# B&R Automation Studio project automationLearning
Automation Studio 4.9

## Configuration MirUnitTest

CPU X20CP0484, AutomationRuntime 6.0.2, Build 11.3.0, Vc 6.0.0

### Hardware
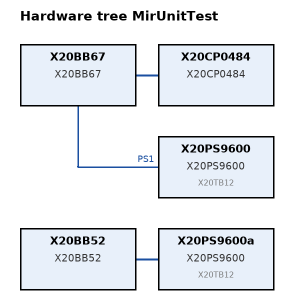
```
X20BB52 : X20BB52 v1.2.0.0
X20BB67 : X20BB67 v1.3.0.0
X20CP0484 : X20CP0484 v1.8.1.0  [SL -> X20BB67.SL1]
  TimerDeviceType = SWIOTIMER
  Cyclic1Duration = 10000
  Cyclic1Tolerance = 10000
  Cyclic2Duration = 20000
  Cyclic2Tolerance = 20000
  Cyclic3Duration = 50000
  Cyclic3Tolerance = 50000
  Cyclic4Duration = 100000
  Cyclic4Tolerance = 100000
  Cyclic5Duration = 200000
  Cyclic5Tolerance = 200000
  Cyclic6Duration = 500000
  Cyclic6Tolerance = 500000
  Cyclic7Duration = 1000000
  Cyclic7Tolerance = 1000000
  Cyclic8Duration = 10000
  Cyclic8Tolerance = 30000000
  FileDevice1
  FileDeviceName1 = USER
  FileDevicePath1 = USER_PATH
X20PS9600 : X20PS9600 v1.6.2.0  [PS -> X20BB67.PS1; SS1 -> X20TB12.SS]
X20PS9600a : X20PS9600 v1.6.2.0  [PS -> X20BB52.PS1; SS1 -> X20TB12a.SS]
X20TB12 : X20TB12 v1.0.0.0
X20TB12a : X20TB12 v1.0.0.0
```

## Configuration Mir_config1

CPU X20CP0484-1, AutomationRuntime 6.0.2, Build 11.3.0, Vc 6.0.0

### Task classes (Cpu.sw)
```
Cyclic#4 (cycle 100000 us, tolerance 100000 us):
  MirValveEx <- MirValveExample.prg
  HMI <- HMI.prg
  MirValveE1 <- MirValveExampleST.prg
Libraries: Valve
```

### Hardware
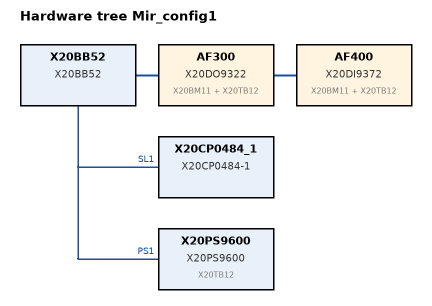
```
AF300 : X20DO9322 v1.6.2.0  [SS1 -> X20TB12a.SS; SL -> X20BM11.SL1]
AF400 : X20DI9372 v1.6.1.0  [SS1 -> X20TB12b.SS; SL -> X20BM11a.SL1]
X20BB52 : X20BB52 v1.2.0.0
  Connector IF6:
    CycleTime = 2000
X20BM11 : X20BM11 v1.1.0.0  [X2X1 -> X20BB52.IF6]
X20BM11a : X20BM11 v1.1.0.0  [X2X1 -> X20BM11.X2X2]
X20CP0484_1 : X20CP0484-1 v1.8.1.0  [SL -> X20BB52.SL1]
  Connector IF2:
    ActivateDevice = 1
  ConfigurationID = Mir_Mir_config1
  Simulation = 1
  TimerDeviceType = SWIOTIMER
  Cyclic1Duration = 10000
  Cyclic1Tolerance = 10000
  Cyclic2Duration = 20000
  Cyclic2Tolerance = 20000
  Cyclic3Duration = 50000
  Cyclic3Tolerance = 50000
  Cyclic4Duration = 100000
  Cyclic4Tolerance = 100000
  Cyclic5Duration = 200000
  Cyclic5Tolerance = 200000
  Cyclic6Duration = 500000
  Cyclic6Tolerance = 500000
  Cyclic7Duration = 1000000
  Cyclic7Tolerance = 1000000
  Cyclic8Duration = 10000
  Cyclic8Tolerance = 30000000
  FileDevice1
  FileDeviceName1 = USER
  FileDevicePath1 = USER_PATH
X20PS9600 : X20PS9600 v1.6.2.0  [PS -> X20BB52.PS1; SS1 -> X20TB12.SS]
X20TB12 : X20TB12 v1.0.0.0
X20TB12a : X20TB12 v1.0.0.0
X20TB12b : X20TB12 v1.0.0.0
```

### IoMap.iom - X20CP0484_1/IoMap.iom
```iecst
VAR_CONFIG
	::gValves.HV_1.cmd_out AT %QX."AF300".DigitalOutput01;
END_VAR
```

## Logical view

Binary libraries used (declarations not repeated): operator, runtime, AsIecCon, astime

### Package Logical/Libraries - Global libraries

### Library Logical/Libraries/MirLib (IEC)

#### Valve_on_off.fbd
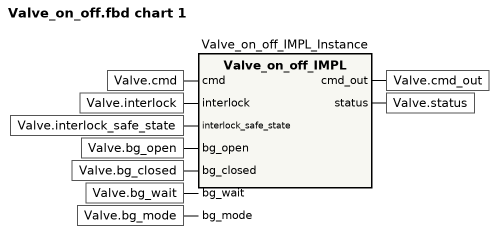
Diagram, in the editor's own instruction-list form stored in the file:
```il
FUNCTION_BLOCK Valve_on_off

{NetworkNumber := 1}
LD Valve.cmd
ST Valve_on_off_IMPL_Instance.cmd
LD Valve.interlock
ST Valve_on_off_IMPL_Instance.interlock
LD Valve.interlock_safe_state
ST Valve_on_off_IMPL_Instance.interlock_safe_state
LD Valve.bg_open
ST Valve_on_off_IMPL_Instance.bg_open
LD Valve.bg_closed
ST Valve_on_off_IMPL_Instance.bg_closed
LD Valve.bg_wait
ST Valve_on_off_IMPL_Instance.bg_wait
LD Valve.bg_mode
ST Valve_on_off_IMPL_Instance.bg_mode
CAL Valve_on_off_IMPL_Instance
LD Valve_on_off_IMPL_Instance.cmd_out
ST Valve.cmd_out
LD Valve_on_off_IMPL_Instance.status
ST Valve.status

END_FUNCTION_BLOCK
```

#### Types.typ - Exported data types
```iecst
TYPE
	bg_expected_enum :
		(
		BG_EXPECTED_OPEN := 0,
		BG_EXPECTED_CLOSED := 1
		);
	limit_switch_mode_enum :
		(
		BG_NONE := 0,
		BG_BOTH := 1,
		BG_OPEN := 2,
		BG_CLOSED := 3
		);
	valve_error_enum :
		(
		NONE := 0,
		TIMEOUT_OPENING := 1,
		TIMEOUT_CLOSING := 2,
		UNEXPECTED_CLOSED := 3,
		UNEXPECTED_OPEN := 4,
		BOTH_FEEDBACK := 5,
		NO_FEEDBACK := 6
		);
	valve_position_enum :
		(
		UNKNOWN := 0,
		CLOSED := 1,
		OPEN := 2,
		INTERMEDIATE := 3
		);
	valve_state_enum :
		(
		OK := 0,
		INTERLOCKED := 1,
		SUPERVISING := 2,
		ERROR := 3
		);
	valve_status_typ : 	STRUCT
		position : valve_position_enum;
		error : valve_error_enum;
		state : valve_state_enum;
	END_STRUCT;
	valve_typ : 	STRUCT
		cmd : BOOL;
		cmd_out : BOOL;
		interlock_safe_state : BOOL;
		status : valve_status_typ;
		interlock : BOOL;
		bg_closed : BOOL;
		bg_open : BOOL;
		bg_wait : TIME;
		bg_mode : limit_switch_mode_enum;
	END_STRUCT;
END_TYPE
```

#### MirLib.fun - Exported functions and function blocks
```iecst
{REDUND_ERROR} FUNCTION_BLOCK Valve_on_off_IMPL (*TODO: Add your comment here*) (*$GROUP=Miro,$CAT=User,$GROUPICON=User.png,$CATICON=User.png*)
	VAR_INPUT
		cmd : {REDUND_UNREPLICABLE} BOOL;
	END_VAR
	VAR_OUTPUT
		cmd_out : BOOL;
	END_VAR
	VAR
		cmd_rising_edge : BOOL;
		cmd_falling_edge : BOOL;
		cmd_changed : BOOL;
		cmd_previous : BOOL;
	END_VAR
	VAR_INPUT
		interlock : BOOL;
		interlock_safe_state : BOOL;
	END_VAR
	VAR
		supervision_active : BOOL;
	END_VAR
	VAR_OUTPUT
		status : valve_status_typ;
	END_VAR
	VAR_INPUT
		bg_open : BOOL; (*Limnit switch for open position*)
		bg_closed : BOOL; (*Limit switch for closed position*)
		bg_wait : TIME;
		bg_mode : limit_switch_mode_enum; (*Limit switch mode*)
	END_VAR
	VAR
		bg_expected_state : bg_expected_enum;
		bg_error : BOOL;
		ElapsedTimer : MirElapsedTimer;
	END_VAR
END_FUNCTION_BLOCK

{REDUND_ERROR} FUNCTION_BLOCK Valve_on_off (*TODO: Add your comment here*) (*$GROUP=User,$CAT=User,$GROUPICON=User.png,$CATICON=User.png*)
	VAR_IN_OUT
		Valve : valve_typ;
	END_VAR
	VAR
		Valve_on_off_IMPL_Instance : Valve_on_off_IMPL;
	END_VAR
END_FUNCTION_BLOCK

{REDUND_ERROR} FUNCTION_BLOCK MirElapsedTimer (*TODO: Add your comment here*) (*$GROUP=User,$CAT=User,$GROUPICON=User.png,$CATICON=User.png*)
	VAR_INPUT
		Enable : {REDUND_UNREPLICABLE} BOOL;
		Delay : TIME;
	END_VAR
	VAR_OUTPUT
		Elapsed : TIME;
		Out : BOOL;
	END_VAR
	VAR
		last_cycle_time : TIME;
		delta_time : TIME;
		cur_time : TIME;
		timer_initialized : BOOL;
	END_VAR
END_FUNCTION_BLOCK
```

#### Valve_on_off_IMPL.st
```iecst
FUNCTION_BLOCK Valve_on_off_IMPL
	ElapsedTimer();
	// RISIGN EDGE OR FALLINH CHECK
	IF cmd = TRUE AND cmd_previous = FALSE THEN
		cmd_rising_edge := TRUE;
		ElapsedTimer.Enable := FALSE;
		bg_error := FALSE;
	ELSE
		cmd_rising_edge := FALSE;
	END_IF;

	IF cmd = FALSE AND cmd_previous = TRUE THEN
		cmd_falling_edge := TRUE;
		ElapsedTimer.Enable := FALSE;
		bg_error := FALSE;
	ELSE
		cmd_falling_edge := FALSE;
	END_IF;

	IF interlock = FALSE THEN ACT_UpdateCmdOut;
	ELSE
		cmd_out := interlock_safe_state;
	END_IF;

	// Handle rising edge
	IF cmd_rising_edge THEN
		CASE bg_mode OF
			BG_NONE:
				// No supervision needed

			BG_BOTH, BG_OPEN:
				ElapsedTimer.Delay := bg_wait;
				ElapsedTimer.Enable := TRUE;
				supervision_active := TRUE;
				bg_expected_state := BG_EXPECTED_OPEN; // Expecting valve to open

			BG_CLOSED:
			// No supervision needed
		END_CASE;
	END_IF;

	// Handle falling edge
	IF cmd_falling_edge THEN
		CASE bg_mode OF
			BG_NONE:
				// No supervision needed
			BG_BOTH, BG_CLOSED:
				ElapsedTimer.Delay := bg_wait;
				ElapsedTimer.Enable := TRUE;
				supervision_active := TRUE;
				bg_expected_state := BG_EXPECTED_CLOSED;

			BG_OPEN:
			// No supervision needed
		END_CASE;
	END_IF;

	// Supervision logic
	IF supervision_active THEN
		CASE bg_mode OF
			BG_BOTH:
				IF (bg_expected_state = BG_EXPECTED_OPEN AND bg_open AND NOT bg_closed) OR
					(bg_expected_state = BG_EXPECTED_CLOSED AND bg_closed AND NOT bg_open) THEN
					supervision_active := FALSE;
					ElapsedTimer.Enable := FALSE;
					bg_error := FALSE;
				END_IF;

			BG_OPEN:
				IF bg_expected_state = BG_EXPECTED_OPEN AND bg_open THEN
					supervision_active := FALSE;
					ElapsedTimer.Enable := FALSE;
					bg_error := FALSE;
				END_IF;

			BG_CLOSED:
				IF bg_expected_state = BG_EXPECTED_CLOSED AND bg_closed THEN
					supervision_active := FALSE;
					ElapsedTimer.Enable := FALSE;
					bg_error := FALSE;
				END_IF;
		END_CASE;

		IF ElapsedTimer.Out THEN
			bg_error := TRUE;
			supervision_active := FALSE;
			ElapsedTimer.Enable := FALSE;
		END_IF;
	END_IF;

	// Continuous monitoring after successful supervision
	IF NOT supervision_active AND NOT bg_error THEN
		CASE bg_mode OF
			BG_BOTH:
				IF cmd_out AND (NOT bg_open OR bg_closed) THEN
					bg_error := TRUE;
				ELSIF NOT cmd_out AND (bg_open OR NOT bg_closed) THEN
					bg_error := TRUE;
				END_IF;
			BG_OPEN:
				IF cmd_out AND NOT bg_open THEN
					bg_error := TRUE;
				END_IF;
			BG_CLOSED:
				IF NOT cmd_out AND NOT bg_closed THEN
					bg_error := TRUE;
				END_IF;
		END_CASE;
	END_IF;
	ACT_UpdateValveStatus;
	cmd_previous := cmd;
END_FUNCTION_BLOCK
```

#### ACT_UpdateCmdOut.st
```iecst
ACTION ACT_UpdateCmdOut:
	IF cmd = TRUE THEN
		cmd_out := TRUE;
	ELSE
		cmd_out := FALSE;
	END_IF;

END_ACTION
```

#### MirElapsedTimer.st
```iecst
(* TODO: Add your comment here *)
FUNCTION_BLOCK MirElapsedTimer
	IF Enable THEN
		IF NOT timer_initialized THEN
			last_cycle_time := clock_ms();
			Elapsed := T#0ms;
			timer_initialized := TRUE;
		ELSE
			cur_time := clock_ms();
			delta_time := cur_time - last_cycle_time;
			last_cycle_time := cur_time;
			Elapsed := Elapsed + delta_time;
		END_IF;
		IF Elapsed >= Delay THEN
			Out := TRUE;
		END_IF;
	ELSE
		Out := FALSE;
		Elapsed := T#0ms;
		timer_initialized := FALSE;
	END_IF;
END_FUNCTION_BLOCK
```

#### ACT_UpdateValveStatus.st
```iecst
ACTION ACT_UpdateValveStatus:

	CASE bg_mode OF
		BG_BOTH:
			IF bg_open AND NOT bg_closed THEN
				status.position := OPEN;
			ELSIF NOT bg_open AND bg_closed THEN
				status.position := CLOSED;
			ELSIF bg_open AND bg_closed THEN
				status.position := INTERMEDIATE;
			ELSE
				status.position := UNKNOWN;
			END_IF;

		BG_OPEN:
			IF bg_open THEN
				status.position := OPEN;
			ELSE
				status.position := UNKNOWN;
			END_IF;

		BG_CLOSED:
			IF bg_closed THEN
				status.position := CLOSED;
			ELSE
				status.position := UNKNOWN;
			END_IF;

		BG_NONE:
			status.position := UNKNOWN;
	END_CASE;

	// Update main status and error
	IF interlock THEN
		status.state := INTERLOCKED;
		status.error := NONE;

	ELSIF supervision_active THEN
		status.state := SUPERVISING;
		status.error := NONE;

	ELSIF bg_error THEN
		status.state := ERROR;

		IF ElapsedTimer.Out THEN
			IF bg_expected_state = BG_EXPECTED_OPEN THEN
				status.error := TIMEOUT_OPENING;
			ELSE
				status.error := TIMEOUT_CLOSING;
			END_IF;

		ELSIF status.position = INTERMEDIATE THEN
			status.error := BOTH_FEEDBACK;

		ELSIF cmd_out AND status.position = CLOSED THEN
			status.error := UNEXPECTED_CLOSED;

		ELSIF NOT cmd_out AND status.position = OPEN THEN
			status.error := UNEXPECTED_OPEN;

		ELSIF status.position = UNKNOWN AND bg_mode <> BG_NONE THEN
			status.error := NO_FEEDBACK;

		ELSE
			status.error := NONE;
		END_IF;

	ELSE
		status.state := OK;
		status.error := NONE;
	END_IF;
END_ACTION
```

### Library Logical/Libraries/Valve (IEC)

#### Types.typ - Exported data types
```iecst
TYPE
	valve_typ : 	STRUCT
		cmd : BOOL;
		cmd_manual : BOOL;
		cmd_out : BOOL;
		cmd_fallback : BOOL;
		mode : BOOL;
		status : INT;
		interlock : BOOL;
	END_STRUCT;
	Valve_mode_enum :
		(
		E_VALVE_MODE_MANUAL := 0,
		E_VALVE_MODE_AUTO := 1,
		E_VALVE_MODE_REMOTE := 2
		);
END_TYPE
```

#### Valve.fun - Exported functions and function blocks
```iecst
{REDUND_ERROR} FUNCTION_BLOCK Valve_on_off_IMPL (*TODO: Add your comment here*) (*$GROUP=Miro,$CAT=User,$GROUPICON=User.png,$CATICON=User.png*)
	VAR_INPUT
		cmd : {REDUND_UNREPLICABLE} BOOL;
		cmd_manual : {REDUND_UNREPLICABLE} BOOL;
		mode : INT;
		cmd_fallback : BOOL;
		interlock : BOOL;
	END_VAR
	VAR_OUTPUT
		cmd_out : BOOL;
		status : {REDUND_UNREPLICABLE} INT;
	END_VAR
END_FUNCTION_BLOCK

{REDUND_ERROR} FUNCTION_BLOCK Valve_on_off (*TODO: Add your comment here*) (*$GROUP=User,$CAT=User,$GROUPICON=User.png,$CATICON=User.png*)
	VAR_IN_OUT
		Valve : valve_typ;
	END_VAR
	VAR
		Valve_on_off_IMPL_Instance : Valve_on_off_IMPL;
	END_VAR
END_FUNCTION_BLOCK
```

#### Valve_on_off_IMPL.st
```iecst
(* TODO: Add your comment here *)
FUNCTION_BLOCK Valve_on_off_IMPL

	IF interlock = FALSE THEN handle_cmd_act;
	ELSE cmd_out := cmd_fallback;
	END_IF;

END_FUNCTION_BLOCK
```

#### handle_cmd_action.st
```iecst
ACTION handle_cmd_act:
	CASE mode OF
		E_VALVE_MODE_MANUAL:
			IF cmd_manual = TRUE THEN
				cmd_out := TRUE;
			ELSE
				cmd_out := FALSE;
			END_IF;
		E_VALVE_MODE_AUTO:
			IF cmd = TRUE THEN
				cmd_out := TRUE;
			ELSE
				cmd_out := FALSE;
			END_IF;
	END_CASE;
END_ACTION
```

#### Valve_on_off.fbd
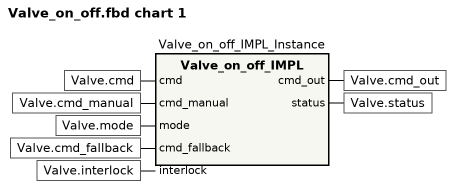
Diagram, in the editor's own instruction-list form stored in the file:
```il
FUNCTION_BLOCK Valve_on_off

{NetworkNumber := 1}
LD Valve.cmd
ST Valve_on_off_IMPL_Instance.cmd
LD Valve.cmd_manual
ST Valve_on_off_IMPL_Instance.cmd_manual
LD Valve.mode
ST Valve_on_off_IMPL_Instance.mode
LD Valve.cmd_fallback
ST Valve_on_off_IMPL_Instance.cmd_fallback
LD Valve.interlock
ST Valve_on_off_IMPL_Instance.interlock
CAL Valve_on_off_IMPL_Instance
LD Valve_on_off_IMPL_Instance.cmd_out
ST Valve.cmd_out
LD Valve_on_off_IMPL_Instance.status
ST Valve.status

END_FUNCTION_BLOCK
```

### Global.typ - Global data types
```iecst
TYPE
	Valves : 	STRUCT
		HV_1 : valve_typ;
		HV_2 : valve_typ;
		HV_3 : valve_typ;
		HV_4 : valve_typ;
		HV_5 : valve_typ;
		HV_7 : valve_typ;
		HV_6 : valve_typ;
	END_STRUCT;
END_TYPE
```

### Global.var - Global variables
```iecst
VAR
	gValves : Valves;
END_VAR
```

### Program Logical/MirValveExampleST (IEC)

#### Variables.var
```iecst
VAR
	HV_1_instance : Valve_on_off;
END_VAR
```

#### Cyclic.st
```iecst
PROGRAM _CYCLIC
	(* Insert code here *)
	 HV_1_instance(Valve := gValves.HV_1);
END_PROGRAM
```

### Program Logical/MirValveExample (IEC)

#### Valve_instanaces.var
```iecst
VAR
	HV_100_FBD : Valve_on_off;
END_VAR
```

#### Cyclic.fbd
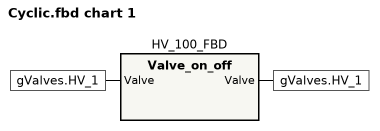
Diagram, in the editor's own instruction-list form stored in the file:
```il
PROGRAM _CYCLIC

{NetworkNumber := 1}
LD gValves.HV_1
ST HV_100_FBD.Valve
CAL HV_100_FBD
LD HV_100_FBD.Valve
ST gValves.HV_1

END_PROGRAM
```

#### Exit.fbd
```iecst
PROGRAM _EXIT

(* TODO : Add your code here *)

END_PROGRAM
```

#### Init.fbd
Diagram, in the editor's own instruction-list form stored in the file:
```il
PROGRAM _INIT

{NetworkNumber := 1}

END_PROGRAM
```

### Program Logical/HMI (IEC)

#### Variables.var
```iecst
VAR
	ctrl : test_ctrl;
	HV_100 : HMI_Valve_on_off;
END_VAR
```

#### Cyclic.st
```iecst
PROGRAM _CYCLIC
	(* Insert code here *)
	IF ctrl.cmd THEN gHV_100.cmd := TRUE;
	ELSE gHV_100.cmd := FALSE;
	END_IF;

	IF ctrl.m0 THEN gHV_100.mode := 0;
	ELSIF ctrl.m1 THEN gHV_100.mode := 1;
	END_IF;
	END_PROGRAM
```

### gValves.var - not listed in the package file held
```iecst
VAR
	gHV_100 : valve_typ;
END_VAR
```

### Program Logical/Timer

#### Variables.var
```iecst
VAR
	test_timer : MirElapsedTimer;
	test_time : TIME;
	MirTimer_0 : MirElapsedTimer;
END_VAR
```

#### Cyclic.st
```iecst
PROGRAM _CYCLIC
	(* Insert code here *)
	MirTimer_0(Delay := T#5s, Enable := TRUE);

	IF MirTimer_0.Elapsed >= T#5s THEN
		 MirTimer_0.Enable := FALSE;
	END_IF;
	test_time := clock_ms();
END_PROGRAM
```

### Valves.typ
```iecst
TYPE
	gValve_collection : 	STRUCT
		HV_1 : valve_typ;
		HV_2 : valve_typ;
		HV_3 : valve_typ;
		HV_4 : valve_typ;
		HV_5 : valve_typ;
		HV_7 : valve_typ;
		HV_6 : valve_typ;
	END_STRUCT;
END_TYPE
```

### Valves.var
```iecst
VAR
	gValves : gValve_collection;
END_VAR
```

### Program Logical/Valves/MirValveExampleST (IEC)

#### Variables.var
```iecst
VAR
	HV_2_instance : Valve_on_off;
	HV_1_instance : Valve_on_off;
END_VAR
```

#### Cyclic.st
```iecst
PROGRAM _CYCLIC
	(* Insert code here *)
	HV_1_instance(Valve := gValves.HV_1);
	HV_2_instance(Valve := gValves.HV_2);
END_PROGRAM
```

### Program Logical/Valves/MirValveExample (IEC)

#### Cyclic.fbd - Cyclic code
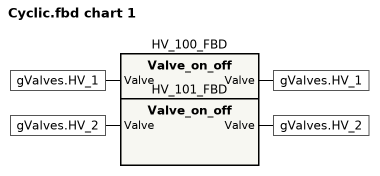
Diagram, in the editor's own instruction-list form stored in the file:
```il
PROGRAM _CYCLIC

{NetworkNumber := 1}
LD gValves.HV_1
ST HV_100_FBD.Valve
CAL HV_100_FBD
LD HV_100_FBD.Valve
ST gValves.HV_1
LD gValves.HV_2
ST HV_101_FBD.Valve
CAL HV_101_FBD
LD HV_101_FBD.Valve
ST gValves.HV_2

END_PROGRAM
```

#### Valve_instanaces.var - Local variables
```iecst
VAR
	HV_100_FBD : Valve_on_off;
	HV_101_FBD : Valve_on_off;
	HV_101_FBD1 : Valve_on_off;
END_VAR
```

### Program Logical/Valves/HMI (IEC)

#### Types.typ
```iecst
TYPE
	HMI_Valve_on_off : 	STRUCT
		cmd : BOOL;
		cmd_manual : BOOL;
		mode : INT;
		status : INT;
	END_STRUCT;
	test_ctrl : 	STRUCT
		cmd : BOOL;
		m1 : BOOL;
		m0 : BOOL;
	END_STRUCT;
END_TYPE
```

#### Variables.var
```iecst
VAR
	HV_100 : HMI_Valve_on_off;
	ctrl : valve_typ;
END_VAR
```

#### Cyclic.st
```iecst
PROGRAM _CYCLIC
    // Map inputs to valve structure
	gValves.HV_1.cmd := ctrl.cmd;
	gValves.HV_1.interlock := ctrl.interlock;
	gValves.HV_1.bg_closed := ctrl.bg_closed;
	gValves.HV_1.bg_open := ctrl.bg_open;
	gValves.HV_1.interlock_safe_state := ctrl.interlock_safe_state;
	gValves.HV_1.bg_wait := ctrl.bg_wait;
	gValves.HV_1.bg_mode := ctrl.bg_mode;

	ctrl.status.error := gValves.HV_1.status.error;
	ctrl.status.position := gValves.HV_1.status.position;
	ctrl.status.state := gValves.HV_1.status.state;
	ctrl.cmd_out := gValves.HV_1.cmd_out;

	END_PROGRAM
```

Listed in the project but not available here: Logical/Libraries/MirLib/Constants.var, Logical/Libraries/Valve/Constants.var, Logical/Valves/MirValveExample/Init.fbd, Logical/Valves/MirValveExample/Exit.fbd, Logical/Valves/MirValveExample/Types.typ
